// TIA Portal V19 export
TYPE "HU_Tank_Config"
// stored: Access Published
   STRUCT
      RecirculationPumpExist : Bool;
      HeatExchangerFanExist : Bool;
      HeatingUnitExistNum : Int;
      ChillerExist : Bool;
      OilMaxTemperature : Real := 70.0;
      WaterMaxTemperature : Real := 60.0;
      TemperatureStartCheckFilters : Real := 35.0;
      HeatingHysteresys : Real := 1.0;
      DelayHeatingStart : Time := T#30S;
      DelayHeatingStop : Time := T#30S;
      DelayCollingStart : Time := T#30S;
      DelayCollingStop : Time := T#30S;
      AnlOilTemp_HighLimit : Real := 100.0;
      AnlOilTemp_LowLimit : Real := 0.0;
      AnlWaterTemp_HighLimit : Real := 100.0;
      AnlWaterTemp_LowLimit : Real := -10.0;
   END_STRUCT;
END_TYPE
